IF (Step(100, TRUE, 'STEP 100')) THEN
    //--------------------------------------------
    StepCompleteWhen(TRUE);
	Messenger.OnCondition(_StepElapsedTime > T#1S).Build().Append('Time is 1s').As().AsInfo();
    //--------------------------------------------		
END_IF;


IF (Step(ErrorStep, TRUE, 'STEP 110')) THEN
    //--------------------------------------------
	;
    //--------------------------------------------		
END_IF;


IF (Step(FinishStep, TRUE, 'SEQUENCE COMPLETE')) THEN
    //--------------------------------------------
	THIS^.CompleteSequence();
    //--------------------------------------------	
END_IF;
END_METHOD

END_FUNCTION_BLOCK

// ---- Template/Component_Cylinder/Base/TcoCylinderBase.TcPOU
FUNCTION_BLOCK ABSTRACT TcoCylinderBase EXTENDS TcoCore.TcoComponent IMPLEMENTS ITcoCylinder
VAR_IN_OUT
	(*~
		<docu>
			<summary>
				Home position sensor.
			</summary>	
		</docu>
	~*)
	{attribute addProperty Name "<#Home position sensor#>"}
	inoAtHomePos : BOOL;
	(*~
		<docu>
			<summary>
				Working position sensor.
			</summary>	
		</docu>
	~*)
	{attribute addProperty Name "<#Work position sensor#>"}
	inoAtWorkPos : BOOL;
END_VAR
VAR_IN_OUT
	(*~
		<docu>
			<summary>
				Move to working home position signal.
			</summary>	
		</docu>
	~*)
	{attribute addProperty Name "<#Move to home position actuator#>"}
	inoToHomePos : BOOL;
	(*~
		<docu>
			<summary>
				Move to working posistion signal.
			</summary>	
		</docu>
	~*)
	{attribute addProperty Name "<#Move to work position actuator#>"}
	inoToWorkPos : BOOL;
END_VAR
VAR
	(*~
		<docu>
			<summary>
				Home position sensor.
			</summary>	
		</docu>
	~*)
	{attribute addProperty Name "<#Home position sensor#>"}
	_atHomePos : BOOL;
	(*~
		<docu>
			<summary>
				Working position sensor.
			</summary>	
		</docu>
	~*)
	{attribute addProperty Name "<#Work position sensor#>"}
	_atWorkPos : BOOL;
	(*~
		<docu>
			<summary>
				Move to working home position signal.
			</summary>	
		</docu>
	~*)
	{attribute addProperty Name "<#Move to home position actuator#>"}
	_toHomePos : BOOL;
	(*~
		<docu>
			<summary>
				Move to working posistion signal.
			</summary>	
		</docu>
	~*)
	{attribute addProperty Name "<#Move to work position actuator#>"}
	_toWorkPos : BOOL;
END_VAR

VAR
	{attribute addProperty Name "<#Home sensor signal#>"}
	_atHomePosSignalInfo : TcoCore.TcoSignalInfo;
	{attribute addProperty Name "<#Work sensor signal#>"}
    _atWorkPosSignalInfo : TcoCore.TcoSignalInfo;
	{attribute addProperty Name "<#Move to home position signal#>"}
    _toHomePosSignalInfo : TcoCore.TcoSignalInfo;
	{attribute addProperty Name "<#Move to work position signal#>"}
    _toWorkPosSignalInfo : TcoCore.TcoSignalInfo;
END_VAR

IF(__ISVALIDREF(inoAtHomePos)) THEN _atHomePos := inoAtHomePos; _atHomePosSignalInfo.GetSignalInfo(SIZEOF(inoAtHomePos), ADR(inoAtHomePos)); END_IF;
IF(__ISVALIDREF(inoAtWorkPos)) THEN _atWorkPos := inoAtWorkPos; _atWorkPosSignalInfo.GetSignalInfo(SIZEOF(inoAtWorkPos), ADR(inoAtWorkPos)); END_IF;
IF(__ISVALIDREF(inoToHomePos)) THEN inoToHomePos := _toHomePos; _toHomePosSignalInfo.GetSignalInfo(SIZEOF(inoToHomePos), ADR(inoToHomePos)); END_IF;
IF(__ISVALIDREF(inoToWorkPos)) THEN inoToWorkPos := _toWorkPos; _toWorkPosSignalInfo.GetSignalInfo(SIZEOF(inoToWorkPos), ADR(inoToWorkPos)); END_IF;

(*~
	<docu>
		<summary>
			Gets whether the piston is in home position. 		
		</summary>			
	</docu>	
~*)
PROPERTY AtHome : bool
GET
AtHome := THIS^._atHomePos;
END_GET
END_PROPERTY

(*~
	<docu>
		<summary>
			Gets whether the piston is in work position. 		
		</summary>			
	</docu>	
~*)
PROPERTY AtWork : bool
GET
AtWork := _atWorkPos;
END_GET
END_PROPERTY

METHOD FB_init : BOOL
VAR_INPUT
	bInitRetains : BOOL; // if TRUE, the retain variables are initialized (warm start / cold start)
	bInCopyCode : BOOL;  // if TRUE, the instance afterwards gets moved into the copy code (online change)
	ParentObject : ITcoObject;	
END_VAR
END_METHOD

(*~
	<docu>
		<summary>
			Gets the `MoveHomeTask` task that controls the moving of the cyclinder in home position.
			<remarks>			
				<note type="important">
					This is an abstract method and must be implemented in derived class.
				</note>
			</remarks>	 		
		</summary>			
	</docu>	
~*)
PROPERTY PUBLIC ABSTRACT MoveHomeTask : TcoCore.ITcoTask
GET
END_GET
END_PROPERTY

(*~
	<docu>
		<summary>
			Starts movement into home position. 		
		</summary>			
	</docu>	
~*)
METHOD MoveToHome : TcoCore.ITcoTaskStatus
IF(MoveHomeTask <> 0) THEN 
	MoveToHome := MoveHomeTask.Invoke();
END_IF;
END_METHOD

(*~
	<docu>
		<summary>
			Starts movement into work position. 		
		</summary>			
	</docu>	
~*)
METHOD MoveToWork :TcoCore.ITcoTaskStatus
IF(MoveWorkTask <> 0) THEN
	MoveToWork := MoveWorkTask.Invoke();
END_IF;
END_METHOD

(*~
	<docu>
		<summary>
			Gets the `MoveWorkTask` task that controls the moving of the cyclinder into work position.
			<remarks>			
				<note type="important">
					This is an abstract method and must be implemented in derived class.
				</note>
			</remarks>	 		
		</summary>			
	</docu>	
~*)
PROPERTY PUBLIC ABSTRACT MoveWorkTask : TcoCore.ITcoTask
GET
END_GET
END_PROPERTY

(*~
	<docu>
		<summary>
			Restore all tasks of this instance into initial state.		 		 		
		</summary>			
	</docu>	
~*)
METHOD  Restore : ITcoRestorable
IF(MoveHomeTask <> 0) THEN MoveHomeTask.Restore(); END_IF;
IF(MoveWorkTask <> 0) THEN MoveWorkTask.Restore(); END_IF;
IF(StopTask <> 0) THEN StopTask.Restore(); END_IF;
END_METHOD

METHOD PROTECTED  ServiceMode
END_METHOD

(*~
	<docu>
		<summary>
			Stops cyclinder movement.
		 	<remarks>			
				<note type="important">
					This method switched off the signals for the movement of the piston in both direction.
					However depending on the pnemumatics configuration the movement may contintue if designed in that way.
					THIS IS NOT A SAFETY FUCTION!
				</note>
			</remarks>	 		
		</summary>			
	</docu>	
~*)
METHOD Stop : TcoCore.ITcoTaskStatus
IF(StopTask <> 0) THEN
	Stop := StopTask.Invoke();
END_IF;
END_METHOD

(*~
	<docu>
		<summary>
			Gets the `StopTask` task that controls the stopping cyclinder movement.
			<remarks>			
				<note type="important">
					This is an abstract method and must be implemented in derived class.
				</note>
			</remarks>	 		
		</summary>			
	</docu>	
~*)
PROPERTY PUBLIC ABSTRACT StopTask : TcoCore.ITcoTask
GET
END_GET
END_PROPERTY

END_FUNCTION_BLOCK

// ---- Template/Component_Cylinder/Tasks/TcoCylinderMoveTask.TcPOU
FUNCTION_BLOCK TcoCylinderMoveTask EXTENDS TcoCore.TcoTask
VAR_INPUT
	PositionSensor		   : BOOL;
	MaxTimeToReachPosition : TIME := T#10S;
	TimeToRefill 		   : TIME := T#100MS;
	PositionName		   : STRING(25);
END_VAR
VAR_IN_OUT
	MoveToPositionSignal : BOOL;
	InverseSignal		 : BOOL;	
END_VAR

VAR
	_stringBuilder : TcoCore.StringBuilder;
END_VAR

IF (THIS^.Execute()) THEN
	IF(THIS^.ElapsedTime > MaxTimeToReachPosition) THEN THIS^.Messenger.Warning(_stringBuilder.Clear().Append(PositionName).Append(' sensor not reached yet.').ToString()); END_IF;
	InverseSignal		 := FALSE;
	MoveToPositionSignal := TRUE;
	THIS^.DoneWhen(PositionSensor);	
END_IF

METHOD PUBLIC FB_init : BOOL
VAR_INPUT
	bInitRetains : BOOL; // if TRUE, the retain variables are initialized (warm start / cold start)
	bInCopyCode : BOOL;  // if TRUE, the instance afterwards gets moved into the copy code (online change)
	ParentObject : ITcoObject;	
END_VAR
END_METHOD

(*~
	<docu>
		<summary>
			Executes when task is aborted.
		</summary>			
	</docu>	
~*)
METHOD PROTECTED OnAbort
MoveToPositionSignal := FALSE;
END_METHOD

METHOD PROTECTED OnError
END_METHOD

METHOD PROTECTED OnStart
END_METHOD

END_FUNCTION_BLOCK

// ---- Template/Station/Data/ST001_ProcessDataManager.TcPOU
FUNCTION_BLOCK ST001_ProcessDataManager EXTENDS TcoData.TcoDataExchange
VAR
	_data : ST001_ProcessData;
END_VAR

SUPER^();

END_FUNCTION_BLOCK

// ---- Template/Station/ST001_AutomatSequence.TcPOU
FUNCTION_BLOCK ST001_AutomatSequence EXTENDS TcoCore.TcoSequencer
VAR_IN_OUT
	inoComponents : ST001_ComponentsHandler;	
END_VAR
VAR
	_gTimer_1 : Tc2_Standard.TON;
END_VAR

(*~
	<docu>
		<summary>
			Main method of the sequener. Custom code needs to be placed here. The sequencer is executed by call of InstanceName.Run() method.
			This method is abstract, and it must be overridden in derived block.
		</summary>
	</docu>
~*)
METHOD PROTECTED  Main : BOOL
IF(NOT __ISVALIDREF(inoComponents)) THEN
	Messenger.Programming('Invalid reference to inoComponents');
	RETURN;
END_IF


IF(Step(inStepID  			:= 100,
	    inEnabled 			:= TRUE,
	    inStepDescription 	:= '<#LOAD PART INTO FIXTURE#>')) 
THEN
//---------------------------------------	    
	IF(inoComponents.PartPresent.IsTrue) THEN
		THIS^.CompleteStep();		
	END_IF;
//---------------------------------------
END_IF;

IF(Step(inStepID  			:= 200,
	    inEnabled 			:= TRUE,
	    inStepDescription 	:= '<#PRESS START BUTTON TO START OPERATIONS#>')) 
THEN
//---------------------------------------
	IF(inoComponents._startButton.IsTrue) THEN
		THIS^.CompleteStep();		
	END_IF;
//---------------------------------------
END_IF;

IF(Step(inStepID  			:= 300,
	    inEnabled 			:= TRUE,
	    inStepDescription 	:= '<#PRESSING#>')) 
THEN
//---------------------------------------
	_gTimer_1(IN := inoComponents.Press.MoveToWork().Done, PT := T#500MS);
	IF(_gTimer_1.Q) THEN
		THIS^.CompleteStep();		
	END_IF;
//---------------------------------------
END_IF;

IF(Step(inStepID  			:= 400,
	    inEnabled 			:= TRUE,
	    inStepDescription 	:= '<#MOVING PRESS TO HOME POSITION#>')) 
THEN
//---------------------------------------
	IF(inoComponents.Press.MoveToHome().Done) THEN
		THIS^.CompleteStep();		
	END_IF;
//---------------------------------------
END_IF;

IF(Step(inStepID  			:= 500,
	    inEnabled 			:= TRUE,
	    inStepDescription 	:= '<#REMOVE PART FROM THE FIXTURE#>')) 
THEN
//---------------------------------------
	IF(inoComponents.PartPresent.IsFalse) THEN
		THIS^.CompleteStep();		
	END_IF;
//---------------------------------------
END_IF;

IF(Step(inStepID  			:= 600,
	    inEnabled 			:= TRUE,
	    inStepDescription 	:= '<#SAVE DATA#>')) 
THEN
//---------------------------------------
	IF(THIS^.Station^.Settings.Create(ULINT_TO_STRING(Context.RealTimeClock.TickClock())).Done) THEN
		THIS^.CompleteStep();		
	END_IF;
//---------------------------------------
END_IF;

		

IF(Step(inStepID  			:= MaxStepID - 1,
	    inEnabled 			:= TRUE,
	    inStepDescription 	:= '<#OPERATIONS COMPLETED#>')) 
THEN
//---------------------------------------
	CompleteSequence();	
//---------------------------------------
END_IF;
END_METHOD

METHOD PROTECTED OnStateChange
VAR_INPUT
	PreviousState	: INT;
	NewState 		: INT;
END_VAR
IF(NOT __ISVALIDREF(inoComponents)) THEN
	RETURN;
END_IF

inoComponents.Press.Restore();
_gTimer_1(IN := FALSE);
END_METHOD

PROPERTY Station : POINTER TO ST001
GET
VAR
	refStation : POINTER TO ST001;
END_VAR
IF(__QUERYPOINTER(Parent,  refStation)) THEN
	Station := refStation;
END_IF;
END_GET
END_PROPERTY

END_FUNCTION_BLOCK

// ---- Template/Component_Carousell/Base/TcoCarouselBase.TcPOU
FUNCTION_BLOCK ABSTRACT TcoCarouselBase EXTENDS TcoCore.TcoComponent

VAR_IN_OUT
	(*~
		<docu>
			<summary>
				In position sensor.
			</summary>	
		</docu>
	~*)
	inoInPosition : BOOL;
	(*~
		<docu>
			<summary>
				In precise position sensor.
			</summary>	
		</docu>
	~*)
	inoInPrecisePosition : BOOL;
END_VAR
VAR_IN_OUT
	(*~
		<docu>
			<summary>
				Enable turn signal.
			</summary>	
		</docu>
	~*)
	{attribute addProperty Name "<#Enable turn#>"}
	inoEnableTurn : BOOL;
	(*~
		<docu>
			<summary>
				Start turn  signal.
			</summary>	
		</docu>
	~*)
	{attribute addProperty Name "<#Start turn#>"}
	inoStartTurn : BOOL;
END_VAR
VAR

	{attribute addProperty Name "<#In position sensor#>"}
	_inPosition : BOOL;
	{attribute addProperty Name "<#In precise position sensor#>"}
	_inPrecisePosition : BOOL;
	(*~
		<docu>
			<summary>
				Enable turn  signal.
			</summary>	
		</docu>
	~*)
	{attribute addProperty Name "<#Enable turn table#>"}
	_enableTurn : BOOL;
	(*~
		<docu>
			<summary>
				Start trun signal.
			</summary>	
		</docu>
	~*)
	{attribute addProperty Name "<#Start turn table#>"}
	_startTurn : BOOL;
END_VAR

VAR
	{attribute addProperty Name "<#In position signal#>"}
	_InPositionSignalInfo : TcoCore.TcoSignalInfo;
	{attribute addProperty Name "<#In precise position signal#>"}
    _InPrecisePositionSignalInfo : TcoCore.TcoSignalInfo;
	{attribute addProperty Name "<#Enable turn signal#>"}
    _EnableTurnSignalInfo : TcoCore.TcoSignalInfo;
	{attribute addProperty Name "<#Start turn signal#>"}
    _StartTurnSignalInfo : TcoCore.TcoSignalInfo;
END_VAR

IF(__ISVALIDREF(inoInPosition)) THEN _inPosition := inoInPosition; _InPositionSignalInfo.GetSignalInfo(SIZEOF(inoInPosition), ADR(inoInPosition)); END_IF;
IF(__ISVALIDREF(inoInPrecisePosition)) THEN _inPrecisePosition := inoInPrecisePosition; _InPrecisePositionSignalInfo.GetSignalInfo(SIZEOF(inoInPrecisePosition), ADR(inoInPrecisePosition)); END_IF;
IF(__ISVALIDREF(inoEnableTurn)) THEN inoEnableTurn := _enableTurn; _EnableTurnSignalInfo.GetSignalInfo(SIZEOF(inoEnableTurn), ADR(inoEnableTurn)); END_IF;
IF(__ISVALIDREF(inoStartTurn)) THEN inoStartTurn := _startTurn; _StartTurnSignalInfo.GetSignalInfo(SIZEOF(inoStartTurn), ADR(inoStartTurn)); END_IF;

(*~
	<docu>
		<summary>
			Gets whether the carousel is in  position. 		
		</summary>			
	</docu>	
~*)
PROPERTY InPosition : bool
GET
InPosition := _inPosition;
END_GET
END_PROPERTY

(*~
	<docu>
		<summary>
			Gets whether the carousel is in precise position. 		
		</summary>			
	</docu>	
~*)
PROPERTY InPrecisePosition : bool
GET
InPrecisePosition := _inPrecisePosition;
END_GET
END_PROPERTY

(*~
	<docu>
		<summary>
			Restore all tasks of this instance into initial state.		 		 		
		</summary>			
	</docu>	
~*)
METHOD  Restore : ITcoRestorable
IF(TurnTask <> 0) THEN TurnTask.Restore(); END_IF;
END_METHOD

METHOD PROTECTED  ServiceMode
END_METHOD

(*~
	<docu>
		<summary>
			Starts movement into work position. 		
		</summary>			
	</docu>	
~*)
METHOD Turn :TcoCore.ITcoTaskStatus
IF(TurnTask <> 0) THEN
	Turn := TurnTask.Invoke();
END_IF;
END_METHOD

(*~
	<docu>
		<summary>
			Gets the `TrunTask` task that controls the rotation from  position to next position in same direction.
			<remarks>			
				<note type="important">
					This is an abstract method and must be implemented in derived class.
				</note>
			</remarks>	 		
		</summary>			
	</docu>	
~*)
PROPERTY PUBLIC ABSTRACT TurnTask : TcoCore.ITcoTask
GET
END_GET
END_PROPERTY

END_FUNCTION_BLOCK

// ---- Template/Component_Carousell/TcoCarousel.TcPOU
{attribute addProperty _turnTableName "<#Turn#>"}
{attribute addProperty _restoreName "<#Restore#>"}
FUNCTION_BLOCK TcoCarousel EXTENDS TcoCarouselBase
VAR_INPUT
		(*~
		<docu>
			<summary>
				This condition prevents the rotation of the table, possibly due to collisions with cylinders, axes, or other objects.
				Do not use signal from Light Curtain here.
			</summary>	
		</docu>
	~*)
	inSafetyCondition:BOOL;
	(*~
		<docu>
			<summary>
				The coded bites are stored in this word, which is valid for the base position of the carousel.
			</summary>	
		</docu>
	~*)
	inBasePositionNumber:WORD;
	
END_VAR
VAR
    {attribute addProperty Name "|[[1]Attribute_turnTableName]|"}
    _turnTask : TcoTurnTableTask(THIS^);

    {attribute addProperty Name "|[[1]Attribute_restoreName]|"}
    _restoreTask : TcoCore.TcoTask(THIS^);
    {attribute addProperty Name "<#Config#>"}
	_config : TcoCarouselConfig;
	{attribute addProperty Name "<#Status#>"}
	_status : TcoCarouselStatus;
END_VAR
VAR	
	increment: INT;
	_index: INT;	
	{attribute 'hide'}
	_positionsIdentifiersClear : ARRAY[0..20] OF UINT;

	_sb : TcoCore.StringBuilder;
	_basePositionNumber: WORD;
END_VAR

SUPER^( inoInPosition := inoInPosition, inoInPrecisePosition := inoInPrecisePosition, inoEnableTurn := inoEnableTurn, inoStartTurn := inoStartTurn);

_status.CurrentPosition:=	inBasePositionNumber;
_status.InPosition:=_inPosition;
_status.InPrecisePosition:=_inPrecisePosition;
_status.TurnSafetyCondition:=inSafetyCondition;




IF(_config.NumberOfPositions <= 0) THEN
	Messenger.Programming('- <#Parameter number of positions is <= 0. The paremeters must be grater than 0.#>'); 
	RETURN;
END_IF

_status.Positions :=_positionsIdentifiersClear;


IF(_config.OffSet = 0) THEN
	_config.OffSet := 1;
END_IF



// Calc position


_status.Positions[_config.NumberOfPositions - 1] := 1+(1 - _config.Offset + _status.CurrentPosition) MOD _config.NumberOfPositions;
FOR _index := 1 TO UINT_TO_INT(_config.NumberOfPositions) - 1 DO	
	_status.Positions[UINT_TO_INT(_config.NumberOfPositions) - 1 - _index] := 1 + ((_status.Positions[UINT_TO_INT(_config.NumberOfPositions) - _index]) MOD (_config.NumberOfPositions));			
END_FOR



// Disables mutualy exclusive actions		
_turnTask.Enabled := NOT _restoreTask.Busy;
	
_turnTask(
	inSafetyCondition:=inSafetyCondition , 
	inoInPosition:=_inPosition , 
	inoInPrecisePosition:=_inPrecisePosition , 
	inoEnableTurn:=_enableTurn , 
	inoStartTurn:=_startTurn , 
	inoConfig:=_config , 
	inoStatus:=_status );


_restoreTask.Enabled:=TRUE;

IF (_restoreTask.Execute()) THEN
 	Restore();

    _restoreTask.DoneWhen(TRUE);
END_IF

// For further discussion about Status
IF(_turnTask.Busy) THEN
	_status.ActionDescription := 'Roatating table to next position ';

ELSIF(_restoreTask.Busy) THEN
	_status.ActionDescription := 'Restoring';
ELSE	
	_status.ActionDescription := 'Idle';
END_IF

SUPER^(inoInPosition := inoInPosition, inoInPrecisePosition := inoInPrecisePosition, inoEnableTurn := inoEnableTurn, inoStartTurn := inoStartTurn);

(*~
	<docu>
		<summary>
			Aborts the turning when the condition is 'true'.
		</summary>
		<remarks>			
				<note type="warning">
					The call of this method will be effective only when called AFTER the initialization of the instance of given TcoCarousel.
				</note>
		</remarks>	
	</docu>
~*)
METHOD Abort : BOOL
VAR_IN_OUT
	(*~
		<docu>
			<summary>
				Condition to abort the turning of the carousel.
			</summary>	
		</docu>
	~*)
	inoDisableCondition : BOOL;
END_VAR
VAR_INPUT
	(*~
		<docu>
			<summary>
				Condition to abort the movement of the carousel can be inverted by this parameter.
			</summary>	
		</docu>
	~*)
	Invert:BOOL;
END_VAR
VAR
	_signalInfo : TcoSignalInfo;
END_VAR
IF ( _turnTask.Busy) AND inoDisableCondition AND NOT Invert THEN
	_signalInfo.GetSignalInfo(SIZEOF(inoDisableCondition), ADR(inoDisableCondition));
	Messenger.Build().Append('<#Turning table aborted due to#> : ').Append(_signalInfo.SymbolPath).As().AsError().Pin();
	_startTurn := FALSE;
	_enableTurn := FALSE;
	IF(__ISVALIDREF(THIS^.inoStartTurn)) THEN THIS^.inoStartTurn := FALSE; END_IF;
	IF(__ISVALIDREF(THIS^.inoEnableTurn)) THEN THIS^.inoEnableTurn := FALSE; END_IF;
	_turnTask.Abort();
ELSIF ( _turnTask.Busy) AND inoDisableCondition AND Invert THEN
	_signalInfo.GetSignalInfo(SIZEOF(inoDisableCondition), ADR(inoDisableCondition));
	Messenger.Build().Append('<#Turning table aborted due to NOT #> : ').Append(_signalInfo.SymbolPath).As().AsError().Pin();
	_startTurn := FALSE;
	_enableTurn := FALSE;
	IF(__ISVALIDREF(THIS^.inoStartTurn)) THEN THIS^.inoStartTurn := FALSE; END_IF;
	IF(__ISVALIDREF(THIS^.inoEnableTurn)) THEN THIS^.inoEnableTurn := FALSE; END_IF;
	_turnTask.Abort();
END_IF
END_METHOD

(*~
	<docu>
		<summary>
			Gets the `StopTask` task that controls the stopping the turning carousel. 		
		</summary>			
	</docu>	
~*)
PROPERTY AbortTask : TcoCore.ITcoTask
GET
AbortTask := _restoreTask;
END_GET
END_PROPERTY

PROPERTY Config : REFERENCE TO TcoCarouselConfig
GET
Config REF= _config;
END_GET
END_PROPERTY

METHOD PUBLIC GetIdentifierAtPosition : UINT
VAR_INPUT
	inPosition:UINT;
END_VAR
GetIdentifierAtPosition:=_turnTask.GetIdentifierAtPosition(inPosition:=inPosition,inPositions:=_status.Positions);
END_METHOD

(*~
	<docu>
		<summary>
			Restore all tasks of this instance into initial state.		 		 		
		</summary>			
	</docu>	
~*)
METHOD  Restore : ITcoRestorable
_turnTask.Restore();
_restoreTask.Abort();
_restoreTask.Restore();
_enableTurn := FALSE;
_startTurn := FALSE;
Messenger.UnPin();
END_METHOD

PROPERTY Status : REFERENCE TO TcoCarouselStatus
GET
Status REF= _status;
END_GET
END_PROPERTY

(*~
	<docu>
		<summary>
			Suspend the turning to next position when the condition is 'true'. Task is still bussy
		</summary>
		<remarks>			
				<note type="warning">
					The call of this method will be effective only when called AFTER the initialization of the instance of given TcoCarousel.
				</note>
		</remarks>	
	</docu>
~*)
METHOD Suspend : BOOL
VAR_IN_OUT
	(*~
		<docu>
			<summary>
				Condition to suspend the movement of the carousel.
			</summary>	
		</docu>
	~*)
	inoDisableCondition : BOOL;
END_VAR
VAR_INPUT
	(*~
		<docu>
			<summary>
				Condition to suspend the movement of the carousel can be inverted by this parameter.
			</summary>	
		</docu>
	~*)
	Invert:BOOL;
END_VAR
VAR
	_signalInfo : TcoSignalInfo;
END_VAR

IF (_turnTask.Busy OR _startTurn OR _enableTurn ) AND inoDisableCondition AND NOT Invert THEN
	_signalInfo.GetSignalInfo(SIZEOF(inoDisableCondition), ADR(inoDisableCondition));
	Messenger.Warning(_sb.Clear().Append('<#Turning table is suspended due to#> : ').Append(_signalInfo.SymbolPath).ToString());
	_startTurn := FALSE;
	_enableTurn := FALSE;
	IF(__ISVALIDREF(THIS^.inoStartTurn)) THEN THIS^.inoStartTurn := FALSE; END_IF;
	IF(__ISVALIDREF(THIS^.inoEnableTurn)) THEN THIS^.inoEnableTurn := FALSE; END_IF;
ELSIF (_turnTask.Busy OR _startTurn OR _enableTurn ) AND inoDisableCondition AND  Invert THEN
	_signalInfo.GetSignalInfo(SIZEOF(inoDisableCondition), ADR(inoDisableCondition));
	Messenger.Warning(_sb.Clear().Append('<#Turning table is suspended due to NOT #> : ').Append(_signalInfo.SymbolPath).ToString());
	_startTurn := FALSE;
	_enableTurn := FALSE;
	IF(__ISVALIDREF(THIS^.inoStartTurn)) THEN THIS^.inoStartTurn := FALSE; END_IF;
	IF(__ISVALIDREF(THIS^.inoEnableTurn)) THEN THIS^.inoEnableTurn := FALSE; END_IF;

END_IF
END_METHOD

(*~
	<docu>
		<summary>
			Gets the `TurnTask` task that controls the moving of the carousel to next position. 		
		</summary>			
	</docu>	
~*)
PROPERTY TurnTask : TcoCore.ITcoTask
GET
TurnTask := _turnTask;
END_GET
END_PROPERTY

END_FUNCTION_BLOCK

// ---- Utilities/Component/FB_ComponentPool.TcPOU
FUNCTION_BLOCK FB_ComponentPool
VAR	
	/// component name
	sName						: STRING;
	
	/// component enable flag
	bEnable						: BOOL := FALSE;
	
	/// component state
	eState						: E_ComponentState;	
	
	/// Area
	eMachineArea				: E_MachineArea;	
	                			

		
	aComponents					: ARRAY[0..COMP.nMaxComponents] OF ITF_Component;
	nComponent					: INT := -1;	

	nErrComponent				: INT;
	sErrComponentName			: STRING;
	
	
	/// Interfaces  	
	itfEventLog					: ITF_EventLog;
	
END_VAR

///
/// 
/// HF/www.asma.at/02.2022
///

/// Get's or set's a value indicating whether this component is active or not.
PROPERTY EnablePool : BOOL
GET
EnablePool := bEnable;
END_GET
SET
VAR
	iIdx			: INT;
END_VAR
bEnable := EnablePool;

// run all components
FOR iIdx := 0 TO COMP.nMaxComponents DO
	// chk valid pointer
	IF aComponents[iIdx] <> 0 THEN
		aComponents[iIdx].Enable := EnablePool;
	END_IF
END_FOR
END_SET
END_PROPERTY

METHOD FB_init : BOOL
VAR_INPUT
	bInitRetains : BOOL; // if TRUE, the retain variables are initialized (warm start / cold start)
	bInCopyCode : BOOL;  // if TRUE, the instance afterwards gets moved into the copy code (online change)
END_VAR
itfEventLog := GVL.fbEventLog;
END_METHOD

METHOD GetComponent : POINTER TO FB_Component
VAR_INPUT
	nSubComp			:INT;	
END_VAR

VAR
	ptTmp				: POINTER TO FB_Component;
	bFound				: BOOL;
END_VAR
bFound := __QUERYPOINTER(aComponents[nSubComp], ptTmp);

IF bFound THEN
	GetComponent := ptTmp;
ELSE
	GetComponent := 0;
END_IF
END_METHOD

METHOD GetItfComponent : ITF_Component
VAR_INPUT
	nSubComp			:INT;	
END_VAR
GetItfComponent := aComponents[nSubComp];
END_METHOD

METHOD HaltPool
VAR_INPUT
	StoppCategory					: INT;			// 0...ungesteuertes Stillsetzen     1...gesteuertes Stillsetzen     2...gesteuertes Stillsetzen ohne Trennung der Energiezufuhr							
END_VAR
VAR
	iIdx			: INT;
	itfAxis			: ITFMotionComponent;
	//ptLifting		: POINTER TO FB_LiftingUnit;
END_VAR
// run all components
FOR iIdx := 0 TO COMP.nMaxComponents DO
	// chk valid pointer
	IF aComponents[iIdx] <> 0 THEN
		// chk component is active
		IF NOT aComponents[iIdx].Enable THEN
			CONTINUE;
		END_IF
		
		aComponents[iIdx].Halt(StoppCategory);
		
		
	END_IF
END_FOR
END_METHOD

PROPERTY MachineArea : E_MachineArea
GET
MachineArea := eMachineArea;
END_GET
SET
VAR
	iIdx			: INT;
END_VAR
eMachineArea := MachineArea;

// run all components
FOR iIdx := 0 TO COMP.nMaxComponents DO
	// chk valid pointer
	IF aComponents[iIdx] <> 0 THEN
		aComponents[iIdx].MachineArea := MachineArea;
	END_IF
END_FOR
END_SET
END_PROPERTY

PROPERTY PoolName : STRING
GET
PoolName := sName;
END_GET
SET
sName := PoolName;
END_SET
END_PROPERTY

PROPERTY PoolState : E_ComponentState
GET
PoolState := eState;
END_GET
END_PROPERTY

/// Registrierung von PM Sub-Komponenten.
METHOD RegisterComponent
VAR_INPUT
	sName			: STRING;
	fbComponent  	: ITF_Component;
END_VAR
//IF nComponent = -1 THEN
//	ResetComponents();
//END_IF

IF fbComponent = 0 THEN
	RETURN;
END_IF


// register sub-component
aComponents[nComponent] := fbComponent;
fbComponent.Name := sName;
fbComponent.BMK := CONCAT3(THIS^.sName,' | ',sName);
fbComponent.MachineArea := eMachineArea;
fbComponent.Enable := FALSE;

// increment counter
IF nComponent < COMP.nMaxComponents THEN
	nComponent := nComponent + 1;
ELSE
	eState := E_ComponentState.error;
	RETURN;
END_IF
END_METHOD

METHOD ResetComponents
VAR_INPUT
END_VAR
nComponent := 0;
MEMSET(ADR(aComponents), 0, SIZEOF(aComponents));
eState := E_ComponentState.none;
END_METHOD

METHOD ResetPool
VAR_INPUT
	bOnlyActive			: BOOL;
	bOnlyNotRunning		: BOOL;
	eComponentType		: E_ComponentType;
	eExpectType			: E_ComponentType;
END_VAR

VAR
	iIdx				: INT;
END_VAR
/// reset all components				
FOR iIdx := 0 TO COMP.nMaxComponents DO
	IF aComponents[iIdx] <> 0 THEN
		
		IF aComponents[iIdx].State = E_ComponentState.running AND bOnlyNotRunning THEN
			CONTINUE;
		END_IF
	
		IF bOnlyActive AND NOT aComponents[iIdx].Enable THEN
			CONTINUE;
		END_IF
		
		IF (eComponentType = E_ComponentType.none OR aComponents[iIdx].Typ = eComponentType) AND
		   (eExpectType = E_ComponentType.none OR aComponents[iIdx].Typ <> eExpectType) THEN
			aComponents[iIdx].Reset();		
		END_IF
		
	END_IF
END_FOR
END_METHOD

/// Run component logic
{attribute 'object_name' := 'RunPool'}
METHOD RunPool

VAR
	iIdx			: INT;
END_VAR
// set overall component state, prio:
// 1. E_ComponentState.eComponentState_error		( --> at least one has error)
// 2. E_ComponentState.eComponentState_none			( --> at least one state is not set)
// 3. E_ComponentState.eComponentState_resetting	( --> at least one is rsetting)
// 4. E_ComponentState.eComponentState_ready		( --> at least one is in ready state)
// 5. E_ComponentState.eComponentState_running		( --> all active are running)

// init with running state
eState := E_ComponentState.running;

// run all components
FOR iIdx := 0 TO COMP.nMaxComponents DO
	// chk valid pointer
	IF aComponents[iIdx] <> 0 THEN
		// chk component is active
		IF aComponents[iIdx].Enable THEN
			aComponents[iIdx].Base();
			// run component and get it's state 
			CASE aComponents[iIdx].State OF
				E_ComponentState.error:
					IF nErrComponent = 0 THEN
						nErrComponent := iIdx;
						sErrComponentName := aComponents[iIdx].Name;
					END_IF
					eState := E_ComponentState.error;	
					
				E_ComponentState.none:
					IF eState <> E_ComponentState.error THEN
						eState := E_ComponentState.none;
					END_IF
					
				E_ComponentState.resetting:
					IF eState <> E_ComponentState.error AND eState <> E_ComponentState.none THEN
						eState := E_ComponentState.resetting;
					END_IF
					
				E_ComponentState.ready:
					IF eState = E_ComponentState.running THEN
						eState := E_ComponentState.ready;
					END_IF					
			END_CASE
		END_IF
	END_IF
END_FOR
END_METHOD

END_FUNCTION_BLOCK

// ---- Utilities/Helpers/Concat/Concat3.TcPOU
FUNCTION Concat3 : T_MaxString
VAR_INPUT
	sExpression1: T_maxString;
	sExpression2: T_maxString;
	sExpression3: T_maxString;
END_VAR

Concat3 := CONCAT(sExpression1, sExpression2);
Concat3 := CONCAT(Concat3, sExpression3);

END_FUNCTION

// ---- Utilities/EventLog/Base/FB_LoggingProviderBase.TcPOU
FUNCTION_BLOCK FB_LoggingProviderBase IMPLEMENTS ITFLoggingProvider

/// Add log method
{attribute 'object_name' := 'AddLog'}
METHOD AddLog : BOOL
VAR_INPUT
	/// log message 
	sText: T_MaxString;
	/// log source
	sSource: STRING;
	///	level: eLogLevelNone, eLogLevelError, eLogLevelWarning, eLogLevelInformation	
	eLevel: E_LogLevel;
END_VAR
VAR
	idx: INT;
END_VAR
///
/// Funktionen zum Hinzufuegen einer Log-Nachricht
/// Rueckgabe: TRUE, bei Erfolg, anderenfalls FALSE
/// 17.05.2010		www.rmth.at
///

idx := iLogArraySize;
REPEAT
	arLoggs[idx] := arLoggs[idx - 1];
    idx:= idx - 1;
UNTIL
    	idx = 0
END_REPEAT

arLoggs[0].sText:= sText;
arLoggs[0].sSource:= sSource;
arLoggs[0].bSaveRequest := TRUE;
arLoggs[0].bSaved  := FALSE;
arLoggs[0].eLevel := eLevel;
arLoggs[0].sTime := sTimeString;

//	Return Result
AddLog := TRUE;
END_METHOD

{attribute 'object_name' := 'Run'}
METHOD Run
END_METHOD

END_FUNCTION_BLOCK

// ---- Utilities/Helpers/Color/F_DWORD2CMYK.TcPOU
FUNCTION F_DWORD2CMYK : ST_ColorCMYK
VAR_INPUT
	Color					: DWORD;
END_VAR

VAR
	stColor					: ST_COLOR;
	tmpArray				: ARRAY[0..3] OF BYTE;
	
	Rc						: REAL;
	Gc						: REAL;
	Bc						: REAL;

	K						: REAL;
	
END_VAR

stColor := F_DWORD2RGB(Color);

Rc := stColor.nRed / 255;
Gc := stColor.nGreen / 255;
Bc := stColor.nBlue / 255;

IF (Rc + Gc + Bc) = 0 THEN
	F_DWORD2CMYK.nCyan := 0;
	F_DWORD2CMYK.nMagenta := 0;
	F_DWORD2CMYK.nYellow := 0;
	F_DWORD2CMYK.nKey := 100;	
	RETURN;
END_IF

K := TO_BYTE(1 - MAX(Rc, MAX(Gc, Bc)));

F_DWORD2CMYK.nCyan := TO_BYTE((1-Rc-K)/(1-K));
F_DWORD2CMYK.nMagenta := TO_BYTE((1-Gc-K)/(1-K));
F_DWORD2CMYK.nYellow := TO_BYTE((1-Bc-K)/(1-K));
F_DWORD2CMYK.nKey := TO_BYTE(K);

END_FUNCTION

// ---- Utilities/Helpers/Color/F_RGB2DWORD.TcPOU
FUNCTION F_RGB2DWORD : DWORD
VAR_INPUT
	Color					: ST_Color;
END_VAR

VAR
	tmpArray				: ARRAY[0..3] OF BYTE;
END_VAR

tmpArray[0] := Color.nBlue;
tmpArray[1] := Color.nGreen;
tmpArray[2] := Color.nRed;
tmpArray[3] := 255;

MEMCPY(ADR(F_RGB2DWORD), ADR(tmpArray), SIZEOF(DWORD));

END_FUNCTION

// ---- Utilities/Helpers/Concat/Concat10.TcPOU
FUNCTION Concat10 : T_MaxString
VAR_INPUT
	sExpression1: T_maxString;
	sExpression2: T_maxString;
	sExpression3: T_maxString;
	sExpression4: T_maxString;
	sExpression5: T_maxString;
	sExpression6: T_maxString;
	sExpression7: T_maxString;
	sExpression8: T_maxString;
	sExpression9: T_maxString;
	sExpression10: T_maxString;
END_VAR

Concat10 := CONCAT(sExpression1, sExpression2);
Concat10 := CONCAT(Concat10, sExpression3);
Concat10 := CONCAT(Concat10, sExpression4);
Concat10 := CONCAT(Concat10, sExpression5);
Concat10 := CONCAT(Concat10, sExpression6);
Concat10 := CONCAT(Concat10, sExpression7);
Concat10 := CONCAT(Concat10, sExpression8);
Concat10 := CONCAT(Concat10, sExpression9);
Concat10 := CONCAT(Concat10, sExpression9);
Concat10 := CONCAT(Concat10, sExpression10);

END_FUNCTION

// ---- Utilities/Helpers/Concat/Concat4.TcPOU
FUNCTION Concat4 : T_MaxString
VAR_INPUT
	sExpression1: T_maxString;
	sExpression2: T_maxString;
	sExpression3: T_maxString;
	sExpression4: T_maxString;
END_VAR

Concat4 := CONCAT(sExpression1, sExpression2);
Concat4 := CONCAT(Concat4, sExpression3);
Concat4 := CONCAT(Concat4, sExpression4);

END_FUNCTION

// ---- Utilities/Helpers/Concat/Concat5.TcPOU
FUNCTION Concat5 : T_MaxString
VAR_INPUT
	sExpression1: T_maxString;
	sExpression2: T_maxString;
	sExpression3: T_maxString;
	sExpression4: T_maxString;
	sExpression5: T_maxString;
END_VAR

Concat5 := CONCAT(sExpression1, sExpression2);
Concat5 := CONCAT(Concat5, sExpression3);
Concat5 := CONCAT(Concat5, sExpression4);
Concat5 := CONCAT(Concat5, sExpression5);

END_FUNCTION

// ---- Utilities/Helpers/Concat/Concat6.TcPOU
FUNCTION Concat6 : T_MaxString
VAR_INPUT
	sExpression1: T_maxString;
	sExpression2: T_maxString;
	sExpression3: T_maxString;
	sExpression4: T_maxString;
	sExpression5: T_maxString;
	sExpression6: T_maxString;
END_VAR

Concat6 := CONCAT(sExpression1, sExpression2);
Concat6 := CONCAT(Concat6, sExpression3);
Concat6 := CONCAT(Concat6, sExpression4);
Concat6 := CONCAT(Concat6, sExpression5);
Concat6 := CONCAT(Concat6, sExpression6);

END_FUNCTION

// ---- Utilities/Helpers/Concat/Concat8.TcPOU
FUNCTION Concat8 : T_MaxString
VAR_INPUT
	sExpression1: T_maxString;
	sExpression2: T_maxString;
	sExpression3: T_maxString;
	sExpression4: T_maxString;
	sExpression5: T_maxString;
	sExpression6: T_maxString;
	sExpression7: T_maxString;
	sExpression8: T_maxString;
END_VAR

Concat8 := CONCAT(sExpression1, sExpression2);
Concat8 := CONCAT(Concat8, sExpression3);
Concat8 := CONCAT(Concat8, sExpression4);
Concat8 := CONCAT(Concat8, sExpression5);
Concat8 := CONCAT(Concat8, sExpression6);
Concat8 := CONCAT(Concat8, sExpression7);
Concat8 := CONCAT(Concat8, sExpression8);

END_FUNCTION

// ---- Utilities/Helpers/Concat/Concat9.TcPOU
FUNCTION Concat9 : T_MaxString
VAR_INPUT
	sExpression1: T_maxString;
	sExpression2: T_maxString;
	sExpression3: T_maxString;
	sExpression4: T_maxString;
	sExpression5: T_maxString;
	sExpression6: T_maxString;
	sExpression7: T_maxString;
	sExpression8: T_maxString;
	sExpression9: T_maxString;
END_VAR

Concat9 := CONCAT(sExpression1, sExpression2);
Concat9 := CONCAT(Concat9, sExpression3);
Concat9 := CONCAT(Concat9, sExpression4);
Concat9 := CONCAT(Concat9, sExpression5);
Concat9 := CONCAT(Concat9, sExpression6);
Concat9 := CONCAT(Concat9, sExpression7);
Concat9 := CONCAT(Concat9, sExpression8);
Concat9 := CONCAT(Concat9, sExpression9);

END_FUNCTION

// ---- Utilities/Helpers/Concat/ConcatArray.TcPOU
FUNCTION ConcatArray : T_MaxString
VAR_INPUT
	sArrExpressions: ARRAY[0..15] OF T_maxString;
END_VAR
VAR
	ii: INT;
END_VAR

ConcatArray := '';

FOR ii:=0 TO 15 DO
	ConcatArray := CONCAT(ConcatArray, sArrExpressions[ii]);
END_FOR

END_FUNCTION

// ---- Utilities/Helpers/FB_GetTimeString.TcPOU
FUNCTION_BLOCK FB_GetTimeString
VAR
	fbPulseGetSystemTime: FB_Pulse;
	fbSystemTime: NT_GetTime;
	sTemp: STRING;
	stTimeStruct: TIMESTRUCT;
END_VAR

///
/// Funktion zum Erzeugen eines Zeitstrings
/// 25.04.2006	RE	www.rmth.at
///

sTemp:='';

// read system time
fbPulseGetSystemTime(tPulseTime:=T#100MS);
fbSystemTime(NETID:='', START:=fbPulseGetSystemTime.Q);
fbSystemTime(START:=FALSE);
stTimeStruct:=fbSystemTime.TIMESTR;

IF (stTimeStruct.wYear = 0 AND stTimeStruct.wMonth = 0 AND stTimeStruct.wDay = 0) THEN
	RETURN;
END_IF

(*	date	*)
sTemp:=CONCAT(sTemp , WORD_TO_STRING(stTimeStruct.wYear));

sTemp:=CONCAT(sTemp , '.');
IF stTimeStruct.wMonth < 10 THEN
	sTemp:=CONCAT(sTemp , '0');
END_IF
sTemp:=CONCAT(sTemp , WORD_TO_STRING(stTimeStruct.wMonth));
sTemp:=CONCAT(sTemp , '.');
IF stTimeStruct.wDay < 10 THEN
	sTemp:=CONCAT(sTemp , '0');
END_IF
sTemp:=CONCAT(sTemp , WORD_TO_STRING(stTimeStruct.wDay));

sTemp:=CONCAT(sTemp , '-');

(*	time	*)
IF stTimeStruct.wHour < 10 THEN
	sTemp:=CONCAT(sTemp , '0');
END_IF
sTemp:=CONCAT(sTemp , WORD_TO_STRING(stTimeStruct.wHour));
sTemp:=CONCAT(sTemp , ':');
IF stTimeStruct.wMinute < 10 THEN
	sTemp:=CONCAT(sTemp , '0');
END_IF
sTemp:=CONCAT(sTemp , WORD_TO_STRING(stTimeStruct.wMinute));
sTemp:=CONCAT(sTemp , ':');
IF stTimeStruct.wSecond < 10 THEN
	sTemp:=CONCAT(sTemp , '0');
END_IF
sTemp:=CONCAT(sTemp , WORD_TO_STRING(stTimeStruct.wSecond));
sTemp:=CONCAT(sTemp , ':');
IF stTimeStruct.wMilliseconds < 10 THEN
	sTemp:=CONCAT(sTemp , '00');
ELSIF stTimeStruct.wMilliseconds < 100 THEN
	sTemp:=CONCAT(sTemp , '0');
END_IF
sTemp:=CONCAT(sTemp , WORD_TO_STRING(stTimeStruct.wMilliseconds));

PROPERTY TimeString : STRING
GET
TimeString:=sTemp;
END_GET
END_PROPERTY

END_FUNCTION_BLOCK

// ---- Utilities/Helpers/FB_Pulse.TcPOU
/// Function block plusegenerator for synchron or asynchron duty cycles
FUNCTION_BLOCK FB_Pulse
VAR_INPUT
	/// pulse time total
	tPulseTime: TIME;
	/// duty cycle factor 0 - 1
	///	default value: 0.5 (50% duty cycle)
	fDutyCycle: REAL := 0.5;
END_VAR
VAR_OUTPUT
	Q: BOOL;
END_VAR
VAR
	tonPulse: TON;
END_VAR

///
/// Programm for pulse generators
/// 10.02.2010	TP www.rmth.at
///

tonPulse(IN := NOT tonPulse.Q, PT:=(tPulseTime));
fDutyCycle:=MIN(fDutyCycle, 1);
IF fDutyCycle <= 0 THEN
	Q:=FALSE;
ELSE
	Q := tonPulse.ET <= REAL_TO_TIME((TIME_TO_REAL(tPulseTime) * fDutyCycle));
END_IF

END_FUNCTION_BLOCK

// ---- Utilities/Helpers/FB_TON_RMTH.TcPOU
///
///	Dieser Baustein verzögert ein Signal und gibt positive und negative Flanke dieses Signals aus
///	von Roland Ertl / www.rmth.at / 2009
FUNCTION_BLOCK FB_TON_RMTH
VAR_INPUT
	///	Signal	
	IN: BOOL;
	///	Verzögerungszeit	
	PT: TIME := TIME#100ms;
END_VAR
VAR_OUTPUT
	///	Verzögertes Signal	
	Q: BOOL;
	///	Flanken -> nur für 1 Zyklus aktiv	
	Qr: BOOL;
	///	Flanken -> nur für 1 Zyklus aktiv	
	Qf: BOOL;
END_VAR
VAR
	ton_On: TON;
	rtrig_Pos: R_TRIG;
	ftrig_Neg: F_TRIG;
END_VAR

ton_On(IN:= IN , PT:= PT , Q=> Q , ET=> );
rtrig_Pos(CLK:= ton_On.Q , Q=> Qr );
ftrig_Neg(CLK:= ton_On.Q , Q=> Qf);

END_FUNCTION_BLOCK

// ---- Utilities/Helpers/F_BYTE_TO_INT.TcPOU
FUNCTION F_BYTE_TO_INT : INT
VAR_INPUT
    BY1 : BYTE;
    BY2 : BYTE;
END_VAR
VAR
   OutVAR : WORD; 
   OutVARINT : INT;
END_VAR

OutVar := BY1;
OutVar := SHL(OutVar, 8) OR BY2;

MEMCPY(ADR(OutVARINT), ADR(OutVAR), SIZEOF(INT));

F_BYTE_TO_INT:= OutVARINT;

END_FUNCTION

// ---- Utilities/Helpers/F_GetPlcCycleTime.TcPOU
/// returns the PLC cycle time in seconds for the current task
FUNCTION F_GetPlcCycleTime : LREAL
VAR
	/// cycle time in internal units (parts of 100ns)
	nCycleTime: UDINT;
	/// FB to get the index of the current task 
	fbTaskIndex: GETCURTASKINDEX;
END_VAR

fbTaskIndex();
nCycleTime := TwinCAT_SystemInfoVarList._TaskInfo[fbTaskIndex.index].CycleTime;
F_GetPlcCycleTime := nCycleTime * 1.0E-7;   // Cycle Time is given in parts of 100ns

END_FUNCTION

// ---- Utilities/Helpers/F_GetSystemTime64.TcPOU
/// returns the current system time as a 64 bit integer (one unit is equivalent to 100ns)
FUNCTION F_GetSystemTime64 : ULINT
VAR
	/// lower 32 bit of the current time
	nLow: UDINT;
	/// higher 32 bit of the current time value
	nHigh: UDINT;
	/// FB that returns the current time as 2 x 32 bit 
	fbGetTime: GETSYSTEMTIME;
END_VAR

// get the time
fbGetTime( timeLoDW => nLow, timeHiDW => nHigh );

// build a 64 bit integer 
F_GetSystemTime64 := nHigh;
F_GetSystemTime64 := SHL( F_GetSystemTime64, 32 ) OR nLow;

END_FUNCTION

// ---- Utilities/Helpers/F_TO_STRING.TcPOU
FUNCTION F_TO_STRING : STRING
VAR_INPUT
	Value			: ANY;
END_VAR

VAR
	pWord     : POINTER TO WORD;
END_VAR

IF Value.TypeClass = __SYSTEM.TYPE_CLASS.TYPE_WORD THEN 

	pWord := Value.pValue;
	
	F_TO_STRING := TO_STRING(pWord^);
	
	IF pWord^ < 10 THEN
		CONCAT('0',F_TO_STRING);	
	END_IF

END_IF

END_FUNCTION

// ---- Utilities/Helpers/P_System.TcPOU
/// Program for reading general system informations
PROGRAM P_System
VAR
	fbPulseGetSystemTime: FB_Pulse;
	fbSystemTime: NT_GetTime;
	fbGetTimeString: FB_GetTimeString;
	/// FB to get the index of the current task
	fbTaskIndex: GETCURTASKINDEX;
	iLoopCount: DINT;
	bFirstRun	: BOOL := TRUE;
END_VAR

///
/// Program, für allgemeine Systemprozeduren
/// 03.04.2012	TP	www.rmth.at
///

//	read system time
fbPulseGetSystemTime(tPulseTime:=T#10MS);
fbSystemTime(NETID:=sEmpty, START:=fbPulseGetSystemTime.Q OR bFirstRun);
fbSystemTime(START:=FALSE);

bFirstRun := FALSE;

dtNow := SYSTEMTIME_TO_DT(fbSystemTime.TIMESTR);
fbGetTimeString();
sTimeString := fbGetTimeString.TimeString;

//  read system informations
fbTaskIndex();
stPlcSystemInfo.stPlcAppSystemInfo := TwinCAT_SystemInfoVarList._AppInfo;
stPlcSystemInfo.stPlcTaskSystemInfo := TwinCAT_SystemInfoVarList._TaskInfo[fbTaskIndex.index];
stPlcSystemInfo.fCycleTime := stPlcSystemInfo.stPlcTaskSystemInfo.CycleTime * 1.0E-7;			// Cycle Time is given in parts of [100ns] --> to [s]
stPlcSystemInfo.fLastExecTime := stPlcSystemInfo.stPlcTaskSystemInfo.LastExecTime * 1.0E-7;		// Cycle Time is given in parts of [100ns] --> to [s]

//  create default pulses
iLoopCount		:= (iLoopCount + 1) MOD 100;			// loop
stPulse.bImpulse1000ms	:= (iLoopCount MOD 100) = 1;	// 1000ms impulse
stPulse.bImpulse500ms	:= (iLoopCount MOD 50) = 1; 	// 500ms impulse
stPulse.bImpulse300ms	:= (iLoopCount MOD 30) = 1; 	// 300ms impulse
stPulse.bImpulse200ms	:= (iLoopCount MOD 20) = 1; 	// 200ms impulse
stPulse.bImpulse100ms	:= (iLoopCount MOD 10) = 1; 	// 100ms impulse

IF stPulse.bImpulse1000ms THEN
	stPulse.bToggle1000ms := NOT stPulse.bToggle1000ms;
END_IF

IF stPulse.bImpulse500ms THEN
	stPulse.bToggle500ms := NOT stPulse.bToggle500ms;
END_IF

IF stPulse.bImpulse300ms THEN
	stPulse.bToggle300ms := NOT stPulse.bToggle300ms;
END_IF

IF stPulse.bImpulse200ms THEN
	stPulse.bToggle200ms := NOT stPulse.bToggle200ms;
END_IF

IF stPulse.bImpulse100ms THEN
	stPulse.bToggle100ms := NOT stPulse.bToggle100ms;
END_IF

END_PROGRAM

// ---- Utilities/Sequencer/FB_Sequence.TcPOU
/// Sequence
FUNCTION_BLOCK FB_Sequence

VAR		
	sName				: STRING := 'Aktion';			/// Name of Sequence
	bEnable				: BOOL := TRUE;					/// Enable Sequencer

	/// Sequence
	nSequenceId			: INT;							/// ID of running Sequence
	nNextSequenceId		: INT;							/// ID of next Sequence
	nLastSequenceId		: INT;							/// ID of last Sequence
	nErrorSequenceId	: INT := -1;
	nWaitingSequenceId	: INT := -1;
	
	/// Step
	nStep				: INT;							/// Actual Stepnumber
	nStepMirror			: INT := -1;					/// Copy of Step for first shot trigger
	sClearText			: STRING;						/// Step Description
	nErrorStep			: INT := -1;
	
	/// Commands
	bPause				: BOOL;							/// Pause Sequence only stepping is possible
	bStepping			: BOOL;							/// Single step option
	
	/// Information
	eState				: E_SequenceState;				/// actual Sequence-State
	bFirstShotSequence	: BOOL;							/// actual Sequence first call
	bFirstShotStep		: BOOL;							/// actual Step first call
	bTimeoutStep		: BOOL;							/// Step Timeout - flag 
	sError				: STRING;						/// Error Description
	
	/// Timer
	tMaxStepTime		: TIME := T#0S;					/// maximum Steptime (0 -> infinity)
	tMaxTime			: TIME := T#71582M47S295MS;		/// maximun Time
	tonStep				: TON;							/// Step Timer
	tonStepDelay		: TON;							/// StepDelay Timer
	
	bCondition			: BOOL := TRUE;					/// Condition for Transition
	tDelay				: TIME := T#0S;		
	bAutoNextSequence	: BOOL := TRUE;
	bErrorHandling		: BOOL := FALSE;
	
	/// Process
	nMaxStep			: INT;
	nProgress			: INT := -1;
END_VAR

///
/// Sequence - FB Utility.
/// HF/www.asma.at/02.2018
///

PROPERTY Condition : BOOL
GET
Condition := bCondition;
END_GET
SET
bCondition := Condition;
END_SET
END_PROPERTY

PROPERTY Delay : TIME
GET
Delay := tDelay;
END_GET
SET
tDelay := Delay;
END_SET
END_PROPERTY

PROPERTY Enable : BOOL
GET
Enable := bEnable;
END_GET
SET
bEnable := Enable;
END_SET
END_PROPERTY

PROPERTY EnableAutoNextSequence : BOOL
GET
EnableAutoNextSequence := bAutoNextSequence;
END_GET
SET
bAutoNextSequence := EnableAutoNextSequence;
END_SET
END_PROPERTY

PROPERTY EnableErrorHandling : BOOL
GET
EnableErrorHandling := bErrorHandling;
END_GET
SET
bErrorHandling := EnableErrorHandling;

IF NOT EnableErrorHandling THEN
	nErrorSequenceId := -1;
	nErrorStep := -1;
END_IF
END_SET
END_PROPERTY

PROPERTY ErrorSequenceId : INT
GET
ErrorSequenceId := nErrorSequenceId;
END_GET
SET
	nErrorSequenceId := ErrorSequenceId;
	nErrorStep := -1;
END_SET
END_PROPERTY

PROPERTY ErrorStep : INT
GET
ErrorStep := nErrorStep;
END_GET
SET
	nErrorSequenceId := -1;
	nErrorStep := ErrorStep;
END_SET
END_PROPERTY

PROPERTY ErrorString : STRING
GET
ErrorString := sError;
END_GET
END_PROPERTY

METHOD Finish
VAR_INPUT
END_VAR
nStep := 0;
nStepMirror := -1;
nProgress := -1;

nLastSequenceId := nSequenceId;
nSequenceId := 0;
eState := E_SequenceState.finished;
sError := sEmpty;
END_METHOD

/// aktuelle Sequence wird zum 1. Mal aufgerufen
PROPERTY FirstShotSequence : BOOL
GET
FirstShotSequence := bFirstShotSequence;
END_GET
END_PROPERTY

/// aktueller Schritt wird zum 1. Mal aufgerufen
PROPERTY FirstShotStep : BOOL
GET
FirstShotStep := bFirstShotStep;
END_GET
END_PROPERTY

PROPERTY Info : STRING
GET
Info := sClearText;
END_GET
SET
sClearText := Info;
END_SET
END_PROPERTY

/// Schrittschaltwerk - Initialisierung
METHOD Init
VAR_INPUT
END_VAR
nStep := 0;
nStepMirror := -1;
nProgress := -1;
sError := sEmpty;
tonStepDelay.IN := FALSE;
nNextSequenceId := 0;

nLastSequenceId := nSequenceId;
nSequenceId := 0;
eState := E_SequenceState.none;
END_METHOD

PROPERTY LastSequenceId : INT
GET
LastSequenceId := nLastSequenceId;
END_GET
END_PROPERTY

PROPERTY MaxStep : INT
GET
MaxStep := nMaxStep;
END_GET
SET
nMaxStep := MaxStep;
END_SET
END_PROPERTY

/// Maximale Schirttdauer (0 -> unbegrenzt)
PROPERTY MaxStepTime : TIME
GET
MaxStepTime := tMaxStepTime;
END_GET
SET
tMaxStepTime := MaxStepTime;
END_SET
END_PROPERTY

/// Name der Aktion
PROPERTY Name : STRING
GET
Name := sName;
END_GET
SET
sName := Name;
END_SET
END_PROPERTY

PROPERTY NextSequence : INT
GET
NextSequence := nNextSequenceId;
END_GET
SET
nNextSequenceId := NextSequence;
END_SET
END_PROPERTY

PROPERTY NextSequenceDefined : BOOL
GET
NextSequenceDefined := nNextSequenceId <> 0;
END_GET
END_PROPERTY

/// aktueller Schritt
{attribute 'monitoring' := 'variable'}
PROPERTY NextStep : INT
SET
IF eState = E_SequenceState.finished THEN 
	RETURN;
END_IF

IF bPause THEN
	sClearText := CONCAT('Pause - ', sClearText);
ELSIF NOT Condition THEN
	sClearText := sClearText;
END_IF

tonStepDelay.IN := TRUE;
tonStepDelay.PT:= tDelay;

IF bCondition AND (tDelay = T#0S OR tonStepDelay.Q OR bPause) AND (NOT bPause OR bStepping) THEN
	tonStepDelay(IN := FALSE);
	tDelay := T#0S;
	bCondition := TRUE;
	bStepping := FALSE;
	nStep:= NextStep;
END_IF
END_SET
END_PROPERTY

METHOD Pause 
VAR_INPUT
	Enable			:bool;
END_VAR
bPause := Enable;
END_METHOD

PROPERTY Progress : INT
GET
VAR
	temp			: INT;
END_VAR
IF nSequenceId < 0 THEN
	Progress := -1;
	RETURN;
END_IF

IF eState = E_SequenceState.finished THEN
	Progress := 100;
	RETURN;
END_IF

IF eState <> E_SequenceState.running THEN
	Progress := -1;
	RETURN;
END_IF


nProgress := MAX(nProgress, (nStep * (10000/nMaxStep))/100);

Progress := nProgress;
END_GET
END_PROPERTY

METHOD QueueNext : BOOL
VAR_INPUT
	SequenceId : INT;
END_VAR
nNextSequenceId := SequenceId;
END_METHOD

METHOD Run
// Enabled
IF NOT bEnable THEN
	init();
	RETURN;
END_IF

// Finished
IF eState = E_SequenceState.finished THEN
	sClearText := Concat3('', Name, ' finished');
	eState := E_SequenceState.none;
END_IF
	
// Ready for New - start automatically
IF eState = E_SequenceState.none AND bAutoNextSequence THEN
	IF nNextSequenceId <> 0 THEN
		StartNext();	
	ELSIF nWaitingSequenceId <> -1 THEN
		Start(nWaitingSequenceId);
	END_IF
END_IF

// 1st shot trigger
bFirstShotStep := nStep <> nStepMirror;
bFirstShotSequence := bFirstShotStep AND nStep = 0;
nStepMirror := nStep;

// run timer
tonStep(IN := NOT bFirstShotStep, PT := tMaxTime);
tonStepDelay();

IF bFirstShotStep THEN
	tonStepDelay.IN := FALSE;
END_IF

// step timeout
bTimeoutStep := tMaxStepTime > T#1MS AND tonStep.ET > tMaxStepTime;

// error handling
IF NOT bErrorHandling THEN
	RETURN;
END_IF

// State Error
IF eState = E_SequenceState.error THEN
	
	IF nErrorSequenceId <> -1 THEN
		nSequenceId := nErrorSequenceId;
		nStep := 0;
		nStepMirror := -1;
		eState := E_SequenceState.error_running;
	ELSIF nErrorStep <> -1 THEN
		nStepMirror := nStep;
		nStep := nErrorStep;
		eState := E_SequenceState.error_running;
	END_IF
	
END_IF

// Timeout
IF bTimeoutStep THEN
	eState := E_SequenceState.error;
	sError := Concat7('Timeout: ', sClearText,  '(Sq: ', INT_TO_STRING(nSequenceId), ', Stp: ', INT_TO_STRING(nStep),')');
END_IF
END_METHOD

PROPERTY SequenceId : INT
GET
SequenceId := nSequenceId;
END_GET
END_PROPERTY

METHOD Start
VAR_INPUT
	nId 	: INT;
END_VAR
nStep := 0;
nProgress := -1;
nStepMirror := -1;
//sError := sEmpty;

nSequenceId := nId;
eState := E_SequenceState.running;
bCondition := TRUE;
END_METHOD

METHOD StartLast
VAR_INPUT
END_VAR
IF nLastSequenceId <> 0 THEN
	nStep := 0;
	nProgress := -1;
	nStepMirror := -1;
	//sError := sEmpty;
	
	nSequenceId := nLastSequenceId;
	eState := E_SequenceState.running;
	bCondition := TRUE;
END_IF
END_METHOD

METHOD StartNext
VAR_INPUT
END_VAR
IF nNextSequenceId <> 0 THEN
	nStep := 0;
	nProgress := -1;
	nStepMirror := -1;
	//sError := sEmpty;
	nSequenceId := nNextSequenceId;
	nNextSequenceId := 0;
	
	eState := E_SequenceState.running;
	bCondition := TRUE;
END_IF
END_METHOD

/// aktueller Sequence-Status
PROPERTY State : E_SequenceState
GET
State := eState;
END_GET
END_PROPERTY

/// aktueller Schritt
{attribute 'monitoring' := 'variable'}
PROPERTY Step : INT
GET
Step := nStep;
END_GET
END_PROPERTY

METHOD Stepping
VAR_INPUT
END_VAR
bStepping := TRUE;
END_METHOD

PROPERTY StepTime : Time
GET
StepTime := tonStep.ET;
END_GET
END_PROPERTY

/// Schritt Timeout - flag 
PROPERTY TimeoutStep : BOOL
GET
TimeoutStep := bTimeoutStep;
END_GET
END_PROPERTY

PROPERTY Waiting : BOOL
GET
Waiting := eState = E_SequenceState.waiting;
END_GET
SET
IF Waiting AND eState = E_SequenceState.running THEN
	eState := E_SequenceState.waiting;	
ELSIF NOT Waiting AND eState = E_SequenceState.waiting THEN
	eState := E_SequenceState.running;	
END_IF
END_SET
END_PROPERTY

PROPERTY WaitingSequenceId : INT
GET
WaitingSequenceId := nWaitingSequenceId;
END_GET
SET
nWaitingSequenceId := WaitingSequenceId;
END_SET
END_PROPERTY

END_FUNCTION_BLOCK

// ---- Utilities/Component/Visualisation/Uc_Component.TcVIS
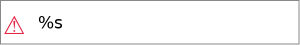
VISUALIZATION Uc_Component  // 300x45
    Rectangle (35,0 265x45), "%s", text variable: stVisu.sName
        p55702900: sel(stvisu.bEnable,colBlack50, colBlack)
    Rectangle (0,5 35x40), "⚠", text variable: stVisu.sName, invisible if: NOT stVisu.bError
        OnMouseClick: execute { stvisu.bReset := TRUE; }
END_VISUALIZATION

// ---- Utilities/EventLog/Visualization/Uc_EventLog.TcVIS
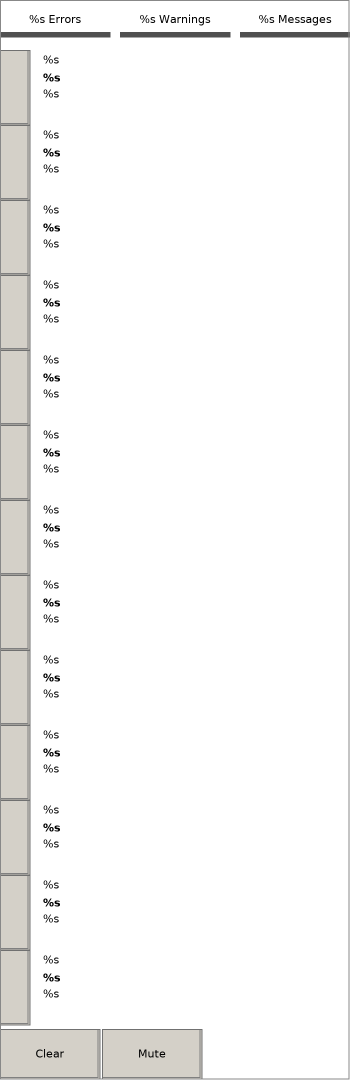
VISUALIZATION Uc_EventLog  // 350x1080
    Frame (0,50 333x977)
        shows Uc_EventLogTable(stVisu := stTable)
    Button (0,1029 100x50), "Clear"
        tap stControl.bQuittAll
    Button (102,1029 100x50), "Mute"
        tap stControl.bMute
    Frame (0,7 350x40)
        shows Uc_EventLogControl(stVisu := stControl)
END_VISUALIZATION

// ---- Utilities/EventLog/Visualization/Uc_EventLogControl.TcVIS
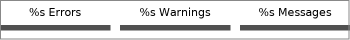
VISUALIZATION Uc_EventLogControl  // 350x40
    Rectangle (0,0 110x25), "%s Errors", text variable: stVisu.nErrorCount
        OnMouseClick: execute { stVisu.bFilterChanged := TRUE; stVisu.bErrorFilter := NOT stVisu.bErrorFilter; }
    Rectangle (0,25 110x5), colour toggle: stVisu.bErrorFilter, colour variable: stVisu.nErrorColor-16#c8000000
        p2167032090: stVisu.nErrorColor
    Rectangle (120,0 110x25), "%s Warnings", text variable: stVisu.nWarningCount
        OnMouseClick: execute { stVisu.bFilterChanged := TRUE; stVisu.bWarningFilter := NOT stVisu.bWarningFilter; }
    Rectangle (240,0 110x25), "%s Messages", text variable: stVisu.nInfoCount
        OnMouseClick: execute { stVisu.bFilterChanged := TRUE; stVisu.bInfoFilter := NOT stVisu.bInfoFilter; }
    Rectangle (120,25 110x5), colour toggle: stVisu.bWarningFilter, colour variable: stVisu.nWarningColor-16#c8000000
        p2167032090: stVisu.nWarningColor
    Rectangle (240,25 110x5), colour toggle: stVisu.bInfoFilter, colour variable: stVisu.nInfoColor-16#c8000000
        p2167032090: stVisu.nInfoColor
END_VISUALIZATION

// ---- Utilities/EventLog/Visualization/Uc_EventLogEntry.TcVIS
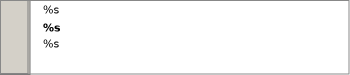
VISUALIZATION Uc_EventLogEntry  // 350x75
    Group (0,0 350x75), invisible if: stVisu.nIdx < 0
        Rectangle (0,0 350x75), colour toggle: stVisu.nIdx = nSelectId
            p2167032090: stVisu.nPriorityColor-16#C8000000
            OnMouseClick: execute { nSelectId := stVisu.nIdx; }
        Rectangle (40,2 300x15), "%s", text variable: stVisu.sRaiseInfo
        Rectangle (40,20 300x16), "%s", text variable: stVisu.sPosition
        Rectangle (40,36 300x32), "%s", text variable: stVisu.sDescription
        Rectangle (0,0 350x75)
            OnMouseClick: execute { nSelectId := stVisu.nIdx; }
        Rectangle (0,0 10x75), colour variable: stVisu.nPriorityColor
            p3450524324: stVisu.nPriorityColor
        Button (0,0 30x75), invisible if: NOT (stVisu.nIdx = nSelectId)
            p2175578022: stVisu.nPriorityColor
            tap bQuit
END_VISUALIZATION

// ---- Utilities/EventLog/Visualization/Uc_EventLogTable.TcVIS
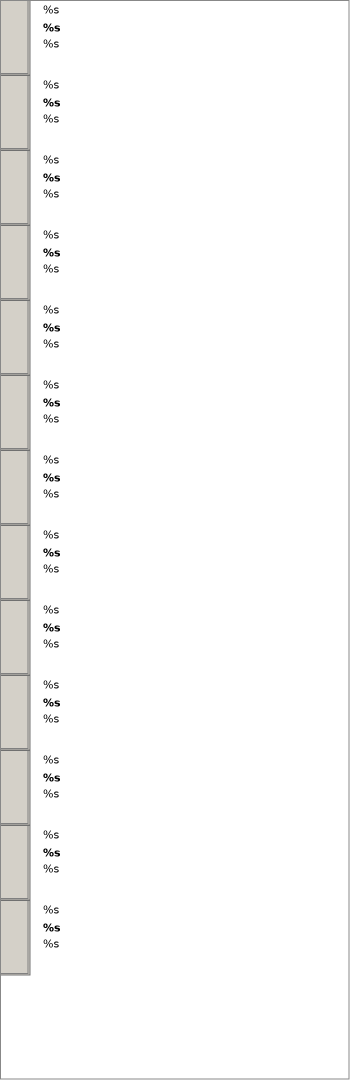
VISUALIZATION Uc_EventLogTable  // 350x1080
    Frame (0,0 350x75)
        shows Uc_EventLogEntry(stVisu := stVisu.astEvents[0], nSelectId := stVisu.nIdx, bQuit := stVisu.bQuitt)
    Frame (0,75 350x75)
        shows Uc_EventLogEntry(stVisu := stVisu.astEvents[1], nSelectId := stVisu.nIdx, bQuit := stVisu.bQuitt)
    Frame (0,150 350x75)
        shows Uc_EventLogEntry(stVisu := stVisu.astEvents[2], nSelectId := stVisu.nIdx, bQuit := stVisu.bQuitt)
    Frame (0,225 350x75)
        shows Uc_EventLogEntry(stVisu := stVisu.astEvents[3], nSelectId := stVisu.nIdx, bQuit := stVisu.bQuitt)
    Frame (0,300 350x75)
        shows Uc_EventLogEntry(stVisu := stVisu.astEvents[4], nSelectId := stVisu.nIdx, bQuit := stVisu.bQuitt)
    Frame (0,375 350x75)
        shows Uc_EventLogEntry(stVisu := stVisu.astEvents[5], nSelectId := stVisu.nIdx, bQuit := stVisu.bQuitt)
    Frame (0,450 350x75)
        shows Uc_EventLogEntry(stVisu := stVisu.astEvents[6], nSelectId := stVisu.nIdx, bQuit := stVisu.bQuitt)
    Frame (0,525 350x75)
        shows Uc_EventLogEntry(stVisu := stVisu.astEvents[7], nSelectId := stVisu.nIdx, bQuit := stVisu.bQuitt)
    Frame (0,600 350x75)
        shows Uc_EventLogEntry(stVisu := stVisu.astEvents[8], nSelectId := stVisu.nIdx, bQuit := stVisu.bQuitt)
    Frame (0,675 350x75)
        shows Uc_EventLogEntry(stVisu := stVisu.astEvents[9], nSelectId := stVisu.nIdx, bQuit := stVisu.bQuitt)
    Frame (0,750 350x75)
        shows Uc_EventLogEntry(stVisu := stVisu.astEvents[10], nSelectId := stVisu.nIdx, bQuit := stVisu.bQuitt)
    Frame (0,825 350x75)
        shows Uc_EventLogEntry(stVisu := stVisu.astEvents[11], nSelectId := stVisu.nIdx, bQuit := stVisu.bQuitt)
    Frame (0,900 350x75)
        shows Uc_EventLogEntry(stVisu := stVisu.astEvents[12], nSelectId := stVisu.nIdx, bQuit := stVisu.bQuitt)
END_VISUALIZATION

// ---- Utilities/List/Visu/Uc_List.TcVIS
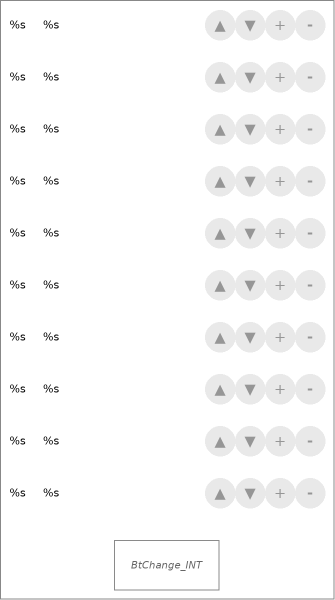
VISUALIZATION Uc_List  // 335x600
    Frame (0,0 335x50)
        shows Uc_Listentry(nId := nIdStartpoint+ 0, stVisu := stVisu)
    Frame (0,52 335x50)
        shows Uc_Listentry(nId := nIdStartpoint+ 1, stVisu := stVisu)
    Frame (0,104 335x50)
        shows Uc_Listentry(nId := nIdStartpoint+ 2, stVisu := stVisu)
    Frame (0,156 335x50)
        shows Uc_Listentry(nId := nIdStartpoint+ 3, stVisu := stVisu)
    Frame (0,208 335x50)
        shows Uc_Listentry(nId := nIdStartpoint+ 4, stVisu := stVisu)
    Frame (0,260 335x50)
        shows Uc_Listentry(nId := nIdStartpoint+ 5, stVisu := stVisu)
    Frame (0,312 335x50)
        shows Uc_Listentry(nId := nIdStartpoint+ 6, stVisu := stVisu)
    Frame (0,364 335x50)
        shows Uc_Listentry(nId := nIdStartpoint+ 7, stVisu := stVisu)
    Frame (0,416 335x50)
        shows Uc_Listentry(nId := nIdStartpoint+ 8, stVisu := stVisu)
    Frame (0,468 335x50)
        shows Uc_Listentry(nId := nIdStartpoint+ 9, stVisu := stVisu)
    Frame (114,540 105x50)
        shows BtChange_INT(Value := nIdStartpoint, minValue := 0, maxValue := 200, stepWidth := 1)
END_VISUALIZATION

// ---- Utilities/List/Visu/Uc_Listentry.TcVIS
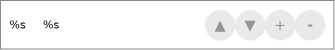
VISUALIZATION Uc_Listentry  // 335x50
    Group (0,0 335x50)
        Rectangle (0,0 335x50), colour toggle: stVisu.nSelected = nId, colour variable: Sel(bAction, colCompBg, colActionColor)
            p2167032090: colButtonDown
            OnMouseClick: execute { stVisu.nSelected := nId; }
            OnMouseDown: execute { bAction := TRUE; colActionColor := colButtonDown; }
            OnMouseEnter: execute { bAction := TRUE; colActionColor := colButtonHover; }
            OnMouseLeave: execute { bAction := FALSE; }
            OnMouseUp: execute { bAction := FALSE; }
        Group (295,10 30x30), text variable: stVisu.bRemove, invisible if: NOT (nId = stVisu.nSelected)
            OnMouseClick: execute { stVisu.nSelected := nId; stVisu.bRemove := TRUE; }
            Ellipse (0,0 30x30)
            Rectangle (0,0 30x30), "-"
        Group (265,10 30x30), text variable: stVisu.bInsert, invisible if: NOT (nId = stVisu.nSelected)
            OnMouseClick: execute { stVisu.nSelected := nId; stVisu.bInsert := TRUE; }
            Ellipse (0,0 30x30)
            Rectangle (0,0 30x30), "+"
        Group (205,10 30x30), text variable: stVisu.bInsert, invisible if: NOT (nId = stVisu.nSelected)
            OnMouseClick: execute { stVisu.nSelected := nId; stVisu.bMoveUp := TRUE; }
            Ellipse (0,0 30x30)
            Rectangle (0,0 30x30), "▲"
        Group (235,10 30x30), text variable: stVisu.bInsert, invisible if: NOT (nId = stVisu.nSelected)
            OnMouseClick: execute { stVisu.nSelected := nId; stVisu.bMoveDown := TRUE; }
            Ellipse (0,0 30x30)
            Rectangle (0,0 30x30), "▼"
        Rectangle (40,0 160x50), "%s", text variable: stVisu.astEntries[nId].sName, colour toggle: stVisu.nSelected = nId, colour variable: Sel(bAction, NormalColor, colActionColor)
            p2167032090: HighlightColor
            p3913753950: textFontName
            OnMouseClick: execute { stVisu.nSelected := nId; }
            OnMouseDown: execute { bAction := TRUE; colActionColor := colButtonDown; }
            OnMouseEnter: execute { bAction := TRUE; colActionColor := colButtonHover; }
            OnMouseLeave: execute { bAction := FALSE; }
            OnMouseUp: execute { bAction := FALSE; }
    Rectangle (0,0 35x50), "%s", text variable: nId, colour toggle: stVisu.nSelected = nId, colour variable: Sel(bAction, NormalColor, colActionColor)
        p2167032090: HighlightColor
        p3913753950: textFontName
        OnMouseClick: execute { stVisu.nSelected := nId; }
        OnMouseDown: execute { bAction := TRUE; colActionColor := colButtonDown; }
        OnMouseEnter: execute { bAction := TRUE; colActionColor := colButtonHover; }
        OnMouseLeave: execute { bAction := FALSE; }
        OnMouseUp: execute { bAction := FALSE; }
END_VISUALIZATION
